TYPE stTransporterVisuSequence :
STRUCT
	//Blocker on Input
	
END_STRUCT
END_TYPE

(* stored: Version 1.1.0.1, ProductVersion 3.1.4024.13
   DUT stTransporterVisuSequence: Id {f6d98f9d-971f-48a5-8733-b9c963d85eff} *)
